(* CODESYS project SPT_Event_Logger.library
   Version: 4.0.0
   Title: SPT Event Logger
   DefaultNamespace: SPT_EventLogger
   Placeholder: SPT Event Logger
   Company: Beckhoff Automation LLC

Project tree, tasks and I/O mapping:
  libraries: Tc2_System, * (Beckhoff Automation GmbH); Tc3_DynamicMemory, * (Beckhoff Automation GmbH); Tc3_EventLogger, 3.3.13.0 (Beckhoff Automation GmbH); Tc3_Module, * (Beckhoff Automation GmbH)
  Alarms/
    function F_ClearAllEventsInClass [ST]
    function F_CreateAllEventsInClass [ST]
    function F_GetMaxSeverityRaised [ST]
    function F_RaiseAlarm [ST]
    function F_RaiseAlarmAndSetFlags [ST]
    function F_RaiseAlarmWithStringParameters [ST]
    function F_RaiseAlarmWithStringsAndFlags [ST]
  Events/
    function block Events [ST]: FB_Exit, FB_Init, CheckEventId, FindActiveSeverity, GetEventInstance, Reset, Arguments, ChangeEventSeverity, ClearEventById, CurrentAlarmSeverity, Name, RaiseEvent, ResetBySeverity
    global variables GVL
  Project Information/
    function F_GetCompany [ST]
    function F_GetTitle [ST]
    function F_GetVersion [ST]
  Version/
    global variables Global_Version
  00000000-0000-0000-0000-000000000000|LICENSE
  LICENSE
*)

// Events/GVL
{attribute 'qualified_only'}
VAR_GLOBAL
	DynamicMemory : FB_DynMem_Manager;
END_VAR

// Version/Global_Version
{attribute 'TcGenerated'}
{attribute 'no-analysis'}
{attribute 'linkalways'}
// This function has been automatically generated from the project information.
VAR_GLOBAL CONSTANT
	{attribute 'const_non_replaced'}
	stLibVersion_SPT_Event_Logger : ST_LibVersion := (iMajor := 4, iMinor := 0, iBuild := 0, iRevision := 0, nFlags := 1, sVersion := '4.0.0');
END_VAR

// Alarms/F_ClearAllEventsInClass
// Initializes event function blocks for an entire event class using auto-generated source info
FUNCTION F_ClearAllEventsInClass
VAR_IN_OUT
	Alarms : ARRAY[*] OF FB_TcAlarm; // Array of Alarms to be defined
END_VAR

VAR
	i : DINT;
END_VAR

FOR i := LOWER_BOUND(Alarms, 1) TO UPPER_BOUND(Alarms, 1) DO
	IF Alarms[i].bRaised THEN
		Alarms[i].Clear(0, 0);
	END_IF
END_FOR

END_FUNCTION

// Alarms/F_CreateAllEventsInClass
// Initializes event function blocks for an entire event class using auto-generated source info
FUNCTION F_CreateAllEventsInClass
VAR_IN_OUT
	Alarms : ARRAY[*] OF FB_TcAlarm; // Array of Alarms to be defined
END_VAR

VAR_INPUT
	ClassSize  : UDINT;					  // Size in bytes of the event class
	pInitEvent : POINTER TO TcEventEntry; // Address of first event in Event Class (Should be the InitReferenceEvent)
	Prefix	   : STRING;				  // String Prefix for the Event Message -- Usually the Module ID and Name
END_VAR

VAR
	i			   : UDINT;
	EventSize	   : UDINT;
	numberOfEvents : UDINT;
	pEvent		   : POINTER TO TcEventEntry;
END_VAR

EventSize	   := SIZEOF(pInitEvent^);
numberOfEvents := ClassSize / EventSize;
FOR i := TO_UDINT(LOWER_BOUND(Alarms, 1)) TO TO_UDINT(UPPER_BOUND(Alarms, 1)) DO
	IF i > numberOfEvents THEN
		EXIT;
	ELSE
		pEvent := pInitEvent + ((i - 1) * EventSize);
		Alarms[i].CreateEx(stEventEntry := pEvent^, 0, 0);
		Alarms[i].ipArguments.AddString(Prefix);
	END_IF
END_FOR

END_FUNCTION

// Alarms/F_GetMaxSeverityRaised
// Compares a collection of alarms to current alarm severity and returns the maximum severity of any raised alarm
FUNCTION F_GetMaxSeverityRaised : TcEventSeverity // Maximum severity
VAR_IN_OUT
	Alarms : ARRAY[*] OF FB_TcAlarm; // Events to compare against
END_VAR

VAR_INPUT
	CurrentSeverity : TcEventSeverity; // Current severity of module alarm
END_VAR

VAR
	i : DINT;
END_VAR

FOR i := LOWER_BOUND(Alarms, 1) TO UPPER_BOUND(Alarms, 1) DO
	IF Alarms[i].bRaised AND (Alarms[i].eSeverity > CurrentSeverity) THEN
		CurrentSeverity := Alarms[i].eSeverity;
	END_IF
END_FOR

F_GetMaxSeverityRaised := CurrentSeverity;

END_FUNCTION

// Events/Events
FUNCTION_BLOCK Events
VAR
	_Name					   : T_MaxString;
	HighestActiveEventSeverity : TcEventSeverity;
	pEventClass				   : PVOID;
	NumberOfEvents			   : UDINT;
	EventBuffer				   : FB_DynMem_Buffer(GVL.DynamicMemory);
	EmptyEvent				   : FB_TcAlarm;
END_VAR

METHOD PUBLIC FB_Exit : BOOL
VAR_INPUT
	bInCopyCode : BOOL; // TRUE: the exit method is called in order to leave the instance which will be copied afterwards (online change).  
END_VAR

VAR
	i		: UDINT;
	ppEvent : POINTER TO POINTER TO FB_TcAlarm;
	pEvent	: POINTER TO FB_TcAlarm;
END_VAR
IF EventBuffer.pBuffer <> 0 THEN
	FOR i := 1 TO NumberOfEvents DO
		ppEvent := EventBuffer.pBuffer + ((i - 1) * SIZEOF(PVOID));
		pEvent	:= ppEvent^;
		pEvent^.Release();
		__DELETE(pEvent);
	END_FOR

	EventBuffer.DeleteBuffer();
END_IF
END_METHOD

METHOD PUBLIC FB_Init : BOOL
VAR_INPUT
	bInitRetains : BOOL; // TRUE: the retain variables are initialized (reset warm / reset cold)
	bInCopyCode	 : BOOL; // TRUE: the instance will be copied to the copy code afterward (online change)
	Name		 : T_MaxString;
	pClass		 : PVOID; // ADR(TC_Events.XY) - TC Event Class in TypeSystem
	nSize		 : UDINT; // SIZEOF(ST_XY) - TC Event Class in TypeSystem
END_VAR

VAR
	i		   : UDINT;
	pEventDef  : POINTER TO TcEventEntry;
	pEvent	   : POINTER TO FB_TcAlarm;
	pBuffer	   : PVOID;
	ppBuffer   : POINTER TO POINTER TO FB_TcAlarm;
	SourceInfo : FB_TcSourceInfo;
END_VAR
FB_Init		   := FALSE;
pEventClass	   := pClass;
NumberOfEvents := nSize / SIZEOF(TcEventEntry);
IF EventBuffer.CreateBuffer(nSize := (NumberOfEvents * SIZEOF(PVOID)), bReset := TRUE) THEN
	IF EventBuffer.bAvailable THEN
		SourceInfo.ResetToDefault();
		SourceInfo.sName := Name;
		FOR i := 1 TO NumberOfEvents DO
			pEvent	  := __NEW(FB_TcAlarm);
			ppBuffer  := EventBuffer.pBuffer + ((i - 1) * SIZEOF(PVOID));
			ppBuffer^ := pEvent;
			pEventDef := pEventClass + ((i - 1) * SIZEOF(TcEventEntry));
			pEvent^.CreateEx2(pEventDef^, SourceInfo);
		END_FOR

		FB_Init := TRUE;
	END_IF
ELSE
	//Buffer not created
END_IF
END_METHOD

METHOD PRIVATE CheckEventId : BOOL
VAR_INPUT
	EventId : UDINT;
END_VAR
CheckEventId := (EventID > 0) AND (EventId <= NumberOfEvents) AND (EventBuffer.bAvailable);
END_METHOD

METHOD PRIVATE FindActiveSeverity
VAR
	i	   : UDINT;
	pEvent : POINTER TO FB_TcAlarm;
END_VAR
HighestActiveEventSeverity := Global.TcEventSeverity.Verbose;
FOR i := 1 TO NumberOfEvents DO
	pEvent := GetEventInstance(i);
	IF (pEvent <> 0) AND_THEN pEvent^.bRaised AND_THEN pEvent^.eSeverity > HighestActiveEventSeverity THEN
		HighestActiveEventSeverity := pEvent^.eSeverity;
	END_IF
END_FOR
END_METHOD

METHOD PRIVATE GetEventInstance : POINTER TO FB_TcAlarm
VAR_INPUT
	EventId : UDINT;
END_VAR

VAR
	ppEvent : POINTER TO POINTER TO FB_TcAlarm;
END_VAR
IF CheckEventId(EventId) THEN
	ppEvent			 := EventBuffer.pBuffer + ((EventId - 1) * SIZEOF(PVOID));
	GetEventInstance := ppEvent^;
ELSE
	GetEventInstance := ADR(EmptyEvent);
END_IF
END_METHOD

METHOD Reset
VAR
	i	   : UDINT;
	pEvent : POINTER TO FB_TcAlarm;
END_VAR
FOR i := 1 TO NumberOfEvents DO
	pEvent := GetEventInstance(i);
	IF (pEvent <> 0) THEN
		pEvent^.Clear();
	END_IF
END_FOR

HighestActiveEventSeverity := Global.TcEventSeverity.Verbose;
END_METHOD

METHOD PUBLIC Arguments : I_TcArguments
VAR_INPUT
	EventId : UDINT;
END_VAR

VAR
	pEvent : POINTER TO FB_TcAlarm;
END_VAR
IF CheckEventId(EventId) THEN
	pEvent := GetEventInstance(EventId);
	IF (pEvent <> 0) THEN
		Arguments := pEvent^.ipArguments;
	ELSE
		Arguments := EmptyEvent.ipArguments;
	END_IF
ELSE
	Arguments := EmptyEvent.ipArguments;
END_IF
END_METHOD

{attribute 'hide'}
METHOD ChangeEventSeverity : BOOL
VAR_INPUT
	EventId	 : UDINT;
	Severity : TcEventSeverity;
END_VAR

VAR
	pEvent	   : POINTER TO FB_TcAlarm;
	EventEntry : TcEventEntry;
	SourceInfo : FB_TcSourceInfo;
	Name	   : STRING;
END_VAR
IF CheckEventId(EventId) THEN
	pEvent := GetEventInstance(EventId);
	IF (pEvent <> 0) THEN
		EventEntry			 := pEvent^.stEventEntry;
		EventEntry.eSeverity := Severity;
		Name				 := pEvent^.ipSourceInfo.sName;
		SourceInfo.ResetToDefault();
		SourceInfo.sName := Name;
		pEvent^.Release();
		pEvent^.CreateEx2(EventEntry, SourceInfo);
	END_IF
END_IF
END_METHOD

METHOD PUBLIC ClearEventById
VAR_INPUT
	EventId : UDINT;
END_VAR

VAR
	pEvent : POINTER TO FB_TcAlarm;
END_VAR
IF CheckEventId(EventId) THEN
	pEvent := GetEventInstance(EventId);
	IF (pEvent <> 0) THEN
		pEvent^.Clear();
	END_IF
END_IF

FindActiveSeverity();
END_METHOD

METHOD CurrentAlarmSeverity : TcEventSeverity
VAR_INPUT
	CurrentSeverity : TcEventSeverity;
END_VAR
IF CurrentSeverity > HighestActiveEventSeverity THEN
	CurrentAlarmSeverity := CurrentSeverity;
	RETURN;
END_IF

CurrentAlarmSeverity := HighestActiveEventSeverity;
END_METHOD

PROPERTY Name : T_MaxString
GET
Name := _Name;
END_GET
SET
_Name := Name;
END_SET
END_PROPERTY

METHOD PUBLIC RaiseEvent
VAR_INPUT
	EventId : UDINT;
END_VAR

VAR
	pEvent : POINTER TO FB_TcAlarm;
END_VAR
IF CheckEventId(EventId) THEN
	pEvent := GetEventInstance(EventId);
	IF (pEvent <> 0) THEN
		IF NOT pEvent^.bRaised THEN
			pEvent^.Raise();
			IF pEvent^.eSeverity > HighestActiveEventSeverity THEN
				HighestActiveEventSeverity := pEvent^.eSeverity;
			END_IF

			pEvent^.ipArguments.Clear();
		END_IF
	END_IF
END_IF
END_METHOD

METHOD ResetBySeverity : BOOL
VAR_INPUT
	Severity : TcEventSeverity;
END_VAR

VAR
	i	   : UDINT;
	pEvent : POINTER TO FB_TcAlarm;
END_VAR
FOR i := 1 TO NumberOfEvents DO
	pEvent := GetEventInstance(i);
	IF (pEvent <> 0) AND_THEN (pEvent^.eSeverity <= Severity) THEN
		pEvent^.Clear();
	END_IF
END_FOR

FindActiveSeverity();
ResetBySeverity := TRUE;
END_METHOD

END_FUNCTION_BLOCK

// Alarms/F_RaiseAlarm
// Raises an alarm and sets fault info to variables which are passed in
FUNCTION F_RaiseAlarm
VAR_IN_OUT
	Alarm : FB_TcAlarm; // Alarm to be raised
END_VAR

IF NOT Alarm.bRaised THEN
	Alarm.Raise(0);
END_IF

END_FUNCTION

// Alarms/F_RaiseAlarmAndSetFlags
// Raises an alarm and sets fault info to variables which are passed in
FUNCTION F_RaiseAlarmAndSetFlags
VAR_IN_OUT
	Alarm	  : FB_TcAlarm; // Alarm to be raised
	ErrorFlag : BOOL;		// Error flag to set (VAR_IN_OUT, put the variable you want the function to SET here)
	ErrorID	  : UDINT;		// Error ID to set (VAR_IN_OUT, put the variable you want the function to SET here) - Will be set using the ID of the given fbAlarm
END_VAR

ErrorFlag := TRUE;
ErrorID	  := Alarm.nEventId;
Alarm.Raise(0);

END_FUNCTION

// Alarms/F_RaiseAlarmWithStringParameters
// Raises an alarm and passes string arguments as parameters for extra fault context/info
FUNCTION F_RaiseAlarmWithStringParameters
VAR_IN_OUT
	Alarm : FB_TcAlarm; // Alarm to be raised
END_VAR

VAR_INPUT
	String_1 : STRING; // First string parameter
	String_2 : STRING; // Second string parameter
	String_3 : STRING; // Third string parameter
END_VAR

Alarm.ipArguments.Clear();
IF String_1 <> '' THEN
	Alarm.ipArguments.AddString(String_1);
END_IF

IF String_2 <> '' THEN
	Alarm.ipArguments.AddString(String_2);
END_IF

IF String_3 <> '' THEN
	Alarm.ipArguments.AddString(String_3);
END_IF

Alarm.Raise(0);

END_FUNCTION

// Alarms/F_RaiseAlarmWithStringsAndFlags
// Raises an alarm and passes string arguments as parameters for extra fault context/info. Additionally sets fault info to variables which are passed in
FUNCTION F_RaiseAlarmWithStringsAndFlags
VAR_IN_OUT
	Alarm	  : FB_TcAlarm; // Alarm to be raised
	ErrorFlag : BOOL;		// Error flag to set (VAR_IN_OUT, put the variable you want the function to SET here)
	ErrorID	  : UDINT;		// Error ID to set (VAR_IN_OUT, put the variable you want the function to SET here) - Will be set using the ID of the given fbAlarm
END_VAR

VAR_INPUT
	String_1 : STRING; // First string parameter
	String_2 : STRING; // Second string parameter
	String_3 : STRING; // Third string parameter
END_VAR

Alarm.ipArguments.Clear();
ErrorFlag := TRUE;
ErrorID	  := Alarm.nEventId;
F_RaiseAlarmWithStringParameters(Alarm	  := Alarm,
								 String_1 := String_1,
								 String_2 := String_2,
								 String_3 := String_3);

END_FUNCTION

// Project Information/F_GetCompany
// This function has been automatically generated from the project information.
{attribute 'signature_flag' := '1073741824'}
{attribute 'TcGenerated'}
{attribute 'no-analysis'}
FUNCTION F_GetCompany : WSTRING
VAR_INPUT
	
END_VAR

F_GetCompany := "Beckhoff Automation LLC";

END_FUNCTION

// Project Information/F_GetTitle
// This function has been automatically generated from the project information.
{attribute 'signature_flag' := '1073741824'}
{attribute 'TcGenerated'}
{attribute 'no-analysis'}
FUNCTION F_GetTitle : WSTRING
VAR_INPUT
	
END_VAR

F_GetTitle := "SPT Event Logger";

END_FUNCTION

// Project Information/F_GetVersion
// This function has been automatically generated from the project information.
{attribute 'signature_flag' := '1073741824'}
{attribute 'TcGenerated'}
{attribute 'no-analysis'}
FUNCTION F_GetVersion : ST_LibVersion
VAR_INPUT
	
END_VAR

F_GetVersion.iMajor := 4;
F_GetVersion.iMinor := 0;
F_GetVersion.iBuild := 0;
F_GetVersion.iRevision := 0;
F_GetVersion.sVersion := '4.0.0';
F_GetVersion.nFlags := 1;

END_FUNCTION
